// TIA Portal V17 export
// export: Created 2024-08-29T18:23:43.1204595Z, ExportSetting WithDefaults, DisplayName Totally Integrated Automation Portal, DisplayVersion V17 Update 7, DisplayName TIA Portal Openness, DisplayVersion V17 Update 7, DisplayName TIA Portal Version Control Interface, DisplayVersion V17, DisplayName SINAMICS Startdrive Advanced, DisplayVersion V17 SP2, DisplayName SINAMICS Startdrive G110M, G120, G120C, G120D, G120P, G115D, DisplayVersion V17 SP2, DisplayName SINAMICS Startdrive G130, G150, S120, S150, SINAMICS MV, S210, DisplayVersion V17 SP2, DisplayName STEP 7 Professional, DisplayVersion V17 Update 7, DisplayName STEP 7 Safety, DisplayVersion V17 Update 6, DisplayName WinCC Advanced / Unified PC, DisplayVersion V17 Update 7
DATA_BLOCK "inputs"   // DB1
{ S7_Optimized_Access := 'TRUE' }
VERSION : 0.1
// stored: AutoNumber false, DBAccessibleFromOPCUA true, DBAccessibleFromWebserver true, IsOnlyStoredInLoadMemory false, IsRetainMemResEnabled false, IsWriteProtectedInAS false, MemoryReserve 100
   VAR RETAIN
      inputSequence : Array[0..32, 0..25] of DInt;   // 32 entradas [modelo, paso]
   END_VAR
   VAR
      activeInputsReq : Array[0..31] of Bool;
   END_VAR
   VAR RETAIN
      maskSequence : Array[0..32, 0..25] of DInt;   // Máscara de entradas
   END_VAR
   VAR
      activeMask : Array[0..31] of Bool;
   END_VAR
   VAR RETAIN
      inputText : Array[0..31] of String;   // Texto HMI de cada entrada
   END_VAR
   VAR
      buttonStatus : Array[0..63] of Bool;
      activeInputsReqDInt : DInt := 131392;   // Estado de sensores en directo
      inputActive : Array[0..31] of Bool;
      euchnerReading : Array[0..254] of Char;
      nestScannerReading : String := '';
      upperScannerReading : String := '';
      nestScanerReceived : Array[0..254] of Char;
      nestScanerReceivedString : String := '';
      upperScannerReceived : Array[0..254] of Char;
      upperScannerReceivedString : String := '';
      euchnerReadingString : String := '$01';
      laserReading : Word := 16#0000;
      laserConstant : Real := 0.0005802801;
      laserReadingInt : DInt := 0;
      readingConversion : LReal := 0.0;
      euchnerName : String := '';
      euchner : Array[0..257] of Byte;
   END_VAR
BEGIN
   inputSequence[0,0] := 23724353;
   inputSequence[0,1] := 827_518_278;
   inputSequence[0,2..4] := 44756294;
   inputSequence[0,5] := 1_252_650_334;
   inputSequence[0,6..7] := 1_118_432_670;
   inputSequence[0,8] := 1_118_432_414;
   inputSequence[0,9] := 44690590;
   inputSequence[0,10] := 44892160;
   inputSequence[0,11..25] := 0;
   inputSequence[1,0] := 23724353;
   inputSequence[1,1] := 827_518_278;
   inputSequence[1,2..4] := 44756294;
   inputSequence[1,5] := 1_252_650_334;
   inputSequence[1,6..7] := 1_118_432_670;
   inputSequence[1,8] := 1_118_432_414;
   inputSequence[1,9] := 44690590;
   inputSequence[1,10] := 44892160;
   inputSequence[1,11..25] := 0;
   inputSequence[2,0] := 23724353;
   inputSequence[2,1] := 827_514_182;
   inputSequence[2,2..4] := 44752198;
   inputSequence[2,5] := 1_252_646_238;
   inputSequence[2,6..7] := 1_118_428_574;
   inputSequence[2,8] := 1_118_428_318;
   inputSequence[2,9] := 44686494;
   inputSequence[2,10] := 44892160;
   inputSequence[2,11..25] := 0;
   inputSequence[3,0] := 23724353;
   inputSequence[3,1] := 827_518_278;
   inputSequence[3,2..4] := 44756294;
   inputSequence[3,5] := 1_252_650_334;
   inputSequence[3,6..8] := 1_118_432_670;
   inputSequence[3,9] := 1_118_432_414;
   inputSequence[3,10] := 44690590;
   inputSequence[3,11] := 44892160;
   inputSequence[3,12..25] := 0;
   inputSequence[4,0] := 23724353;
   inputSequence[4,1] := 827_514_182;
   inputSequence[4,2..4] := 44752198;
   inputSequence[4,5] := 1_252_646_238;
   inputSequence[4,6..7] := 1_118_428_574;
   inputSequence[4,8] := 1_118_428_446;
   inputSequence[4,9] := 1_118_428_318;
   inputSequence[4,10] := 44686494;
   inputSequence[4,11] := 44892160;
   inputSequence[4,12..25] := 0;
   inputSequence[5,0..1] := 64;
   inputSequence[5,2..3] := 128;
   inputSequence[5,4..25] := 0;
   inputSequence[6,0] := 23724353;
   inputSequence[6,1] := 827_780_422;
   inputSequence[6,2] := 44756294;
   inputSequence[6,3] := 44755974;
   inputSequence[6,4] := 1_252_650_334;
   inputSequence[6,5..7] := 1_118_432_670;
   inputSequence[6,8] := 1_118_432_414;
   inputSequence[6,9] := 44630336;
   inputSequence[6,10..25] := 0;
   inputSequence[7,0] := 23724353;
   inputSequence[7,1] := 827_780_422;
   inputSequence[7,2] := 44756294;
   inputSequence[7,3] := 44755974;
   inputSequence[7,4] := 1_252_650_334;
   inputSequence[7,5..7] := 1_118_432_670;
   inputSequence[7,8] := 1_118_432_414;
   inputSequence[7,9] := 44630336;
   inputSequence[7,10..25] := 0;
   inputSequence[8,0] := 23724353;
   inputSequence[8,1] := 827_776_326;
   inputSequence[8,2] := 44752198;
   inputSequence[8,3] := 44751878;
   inputSequence[8,4] := 1_252_646_238;
   inputSequence[8,5] := 1_118_428_574;
   inputSequence[8,6] := 1_118_428_318;
   inputSequence[8,7] := 1_118_428_574;
   inputSequence[8,8] := 1_118_428_318;
   inputSequence[8,9] := 44630336;
   inputSequence[8,10..25] := 0;
   inputSequence[9,0] := 321;
   inputSequence[9,1] := 4193656;
   inputSequence[9,2] := 2_017_459_576;
   inputSequence[9,3] := 1_077_935_482;
   inputSequence[9,4] := 1_073_745_282;
   inputSequence[9,5..6] := 1_073_745_538;
   inputSequence[9,7..9] := 320;
   inputSequence[9,10..25] := 0;
   inputSequence[10,0] := 321;
   inputSequence[10,1] := 4193656;
   inputSequence[10,2] := 2_017_459_576;
   inputSequence[10,3] := 1_077_935_482;
   inputSequence[10,4] := 1_073_745_282;
   inputSequence[10,5..6] := 1_073_745_538;
   inputSequence[10,7..9] := 320;
   inputSequence[10,10..25] := 0;
   inputSequence[11,0] := 321;
   inputSequence[11,1] := 4193656;
   inputSequence[11,2] := 2_017_459_576;
   inputSequence[11,3] := 1_077_935_482;
   inputSequence[11,4] := 1_073_745_282;
   inputSequence[11,5..6] := 1_073_745_538;
   inputSequence[11,7..9] := 320;
   inputSequence[11,10..25] := 0;
   inputSequence[12,0] := 321;
   inputSequence[12,1] := 8387960;
   inputSequence[12,2] := 2_021_653_880;
   inputSequence[12,3] := 1_082_129_786;
   inputSequence[12,4] := 1_077_939_586;
   inputSequence[12,5] := 1_077_939_842;
   inputSequence[12,6] := 1_073_745_538;
   inputSequence[12,7..9] := 320;
   inputSequence[12,10..25] := 0;
   inputSequence[13,0] := 321;
   inputSequence[13,1] := 4193656;
   inputSequence[13,2] := 2_017_459_576;
   inputSequence[13,3] := 1_077_935_482;
   inputSequence[13,4] := 1_073_745_282;
   inputSequence[13,5..6] := 1_073_745_538;
   inputSequence[13,7..9] := 320;
   inputSequence[13,10..25] := 0;
   inputSequence[14,0] := 321;
   inputSequence[14,1] := 4193656;
   inputSequence[14,2] := 2_017_459_576;
   inputSequence[14,3] := 1_077_935_482;
   inputSequence[14,4] := 1_073_745_282;
   inputSequence[14,5..6] := 1_073_745_538;
   inputSequence[14,7..9] := 320;
   inputSequence[14,10..25] := 0;
   inputSequence[15,0] := 11;
   inputSequence[15,1] := 63040522;
   inputSequence[15,2] := 1_338_108_938;
   inputSequence[15,3] := 65137674;
   inputSequence[15,4] := 65135628;
   inputSequence[15,5] := 65134612;
   inputSequence[15,6] := 57344;
   inputSequence[15,7] := 805_363_712;
   inputSequence[15,8] := 10;
   inputSequence[15,9..25] := 0;
   inputSequence[16,0] := 321;
   inputSequence[16,1] := 8387960;
   inputSequence[16,2] := 2_021_653_880;
   inputSequence[16,3] := 1_082_129_786;
   inputSequence[16,4] := 1_077_939_586;
   inputSequence[16,5] := 1_077_939_842;
   inputSequence[16,6] := 1_073_745_538;
   inputSequence[16,7..9] := 320;
   inputSequence[16,10..25] := 0;
   inputSequence[17,0] := 321;
   inputSequence[17,1] := 4193656;
   inputSequence[17,2] := 2_017_459_576;
   inputSequence[17,3] := 1_077_935_482;
   inputSequence[17,4] := 1_073_745_282;
   inputSequence[17,5..6] := 1_073_745_538;
   inputSequence[17,7..9] := 320;
   inputSequence[17,10..25] := 0;
   inputSequence[18,0] := 321;
   inputSequence[18,1] := 4193656;
   inputSequence[18,2] := 2_017_459_576;
   inputSequence[18,3] := 1_077_935_482;
   inputSequence[18,4] := 1_073_745_282;
   inputSequence[18,5..6] := 1_073_745_538;
   inputSequence[18,7..9] := 320;
   inputSequence[18,10..25] := 0;
   inputSequence[19,0] := 321;
   inputSequence[19,1] := 4193656;
   inputSequence[19,2] := 2_017_459_576;
   inputSequence[19,3] := 1_077_935_482;
   inputSequence[19,4] := 1_073_745_282;
   inputSequence[19,5..6] := 1_073_745_538;
   inputSequence[19,7..9] := 320;
   inputSequence[19,10..25] := 0;
   inputSequence[20,0..25] := 0;
   inputSequence[21,0..25] := 0;
   inputSequence[22,0..25] := 0;
   inputSequence[23,0..25] := 0;
   inputSequence[24,0..25] := 0;
   inputSequence[25,0..25] := 0;
   inputSequence[26,0..25] := 0;
   inputSequence[27,0..25] := 0;
   inputSequence[28,0..25] := 0;
   inputSequence[29,0..25] := 0;
   inputSequence[30,0..25] := 0;
   inputSequence[31,0..25] := 0;
   inputSequence[32,0..25] := 0;
   activeInputsReq[0] := TRUE;
   activeInputsReq[1..5] := FALSE;
   activeInputsReq[6] := TRUE;
   activeInputsReq[7] := FALSE;
   activeInputsReq[8] := TRUE;
   activeInputsReq[9..16] := FALSE;
   activeInputsReq[17] := TRUE;
   activeInputsReq[18] := FALSE;
   activeInputsReq[19] := TRUE;
   activeInputsReq[20] := FALSE;
   activeInputsReq[21..22] := TRUE;
   activeInputsReq[23] := FALSE;
   activeInputsReq[24] := TRUE;
   activeInputsReq[25..31] := FALSE;
   maskSequence[0,0] := 66859008;
   maskSequence[0,1] := 66846720;
   maskSequence[0,2] := 66847168;
   maskSequence[0,3..4] := 66846848;
   maskSequence[0,5..8] := 66846720;
   maskSequence[0,9] := 66846862;
   maskSequence[0,10] := 66649232;
   maskSequence[0,11..25] := 0;
   maskSequence[1,0] := 66859008;
   maskSequence[1,1] := 66846720;
   maskSequence[1,2] := 66847168;
   maskSequence[1,3..4] := 66846848;
   maskSequence[1,5..8] := 66846720;
   maskSequence[1,9] := 66846862;
   maskSequence[1,10] := 66649232;
   maskSequence[1,11..25] := 0;
   maskSequence[2,0] := 66859008;
   maskSequence[2,1] := 66846720;
   maskSequence[2,2] := 66847168;
   maskSequence[2,3..4] := 66846848;
   maskSequence[2,5..8] := 66846720;
   maskSequence[2,9] := 66846862;
   maskSequence[2,10] := 66649232;
   maskSequence[2,11..25] := 0;
   maskSequence[3,0] := 66859008;
   maskSequence[3,1] := 66846720;
   maskSequence[3,2] := 66847168;
   maskSequence[3,3..4] := 66846848;
   maskSequence[3,5..7] := 66846720;
   maskSequence[3,8] := 66846976;
   maskSequence[3,9] := 66846720;
   maskSequence[3,10] := 66846848;
   maskSequence[3,11] := 66649232;
   maskSequence[3,12..25] := 0;
   maskSequence[4,0] := 66859008;
   maskSequence[4,1] := 66846720;
   maskSequence[4,2] := 66847168;
   maskSequence[4,3..4] := 66846848;
   maskSequence[4,5..7] := 66846720;
   maskSequence[4,8] := 66847168;
   maskSequence[4,9] := 66846720;
   maskSequence[4,10] := 66846848;
   maskSequence[4,11] := 66649232;
   maskSequence[4,12..25] := 0;
   maskSequence[5,0..1] := -65;
   maskSequence[5,2..3] := -129;
   maskSequence[5,4..25] := 0;
   maskSequence[6,0..2] := 66846720;
   maskSequence[6,3] := 66847168;
   maskSequence[6,4..8] := 66846720;
   maskSequence[6,9] := 66847168;
   maskSequence[6,10..25] := 0;
   maskSequence[7,0..1] := 66846720;
   maskSequence[7,2..3] := 66847168;
   maskSequence[7,4..6] := 66846720;
   maskSequence[7,7] := 66846976;
   maskSequence[7,8] := 66846720;
   maskSequence[7,9] := 66847168;
   maskSequence[7,10..25] := 0;
   maskSequence[8,0..1] := 66846720;
   maskSequence[8,2..3] := 66847168;
   maskSequence[8,4..5] := 66846720;
   maskSequence[8,6..7] := 66846976;
   maskSequence[8,8] := 66846720;
   maskSequence[8,9] := 66847168;
   maskSequence[8,10..25] := 0;
   maskSequence[9,0] := -322;
   maskSequence[9,1] := 2_014_248_960;
   maskSequence[9,2..3] := 983040;
   maskSequence[9,4..5] := 79687736;
   maskSequence[9,6] := 134_213_948;
   maskSequence[9,7..8] := -2;
   maskSequence[9,9] := 134_217_406;
   maskSequence[9,10..25] := 0;
   maskSequence[10,0] := -322;
   maskSequence[10,1] := 2_014_289_920;
   maskSequence[10,2..3] := 1024000;
   maskSequence[10,4..5] := 79687736;
   maskSequence[10,6] := 134_213_948;
   maskSequence[10,7..8] := -2;
   maskSequence[10,9] := 134_217_406;
   maskSequence[10,10..25] := 0;
   maskSequence[11,0] := -322;
   maskSequence[11,1] := 2_014_248_960;
   maskSequence[11,2..3] := 983040;
   maskSequence[11,4..5] := 79687736;
   maskSequence[11,6] := 134_213_948;
   maskSequence[11,7..8] := -2;
   maskSequence[11,9] := 134_217_406;
   maskSequence[11,10..25] := 0;
   maskSequence[12,0] := -322;
   maskSequence[12,1] := 2_014_248_960;
   maskSequence[12,2..3] := 983040;
   maskSequence[12,4..5] := 79687736;
   maskSequence[12,6] := 134_213_948;
   maskSequence[12,7..8] := -2;
   maskSequence[12,9] := 134_217_406;
   maskSequence[12,10..25] := 0;
   maskSequence[13,0] := -322;
   maskSequence[13,1] := 2_014_248_960;
   maskSequence[13,2..3] := 983040;
   maskSequence[13,4..5] := 79687736;
   maskSequence[13,6] := 134_213_948;
   maskSequence[13,7..8] := -2;
   maskSequence[13,9] := 134_217_406;
   maskSequence[13,10..25] := 0;
   maskSequence[14,0] := -322;
   maskSequence[14,1] := 2_014_248_960;
   maskSequence[14,2] := 806_289_408;
   maskSequence[14,3] := 983040;
   maskSequence[14,4..5] := 79687736;
   maskSequence[14,6] := 134_213_948;
   maskSequence[14,7..8] := -2;
   maskSequence[14,9] := 134_217_406;
   maskSequence[14,10..25] := 0;
   maskSequence[15,0] := 0;
   maskSequence[15,1] := 2_080_374_784;
   maskSequence[15,2..3] := 805_306_368;
   maskSequence[15,4..5] := 868_220_928;
   maskSequence[15,6..7] := 268_435_452;
   maskSequence[15,8..25] := 0;
   maskSequence[16,0] := -322;
   maskSequence[16,1] := 2_014_248_960;
   maskSequence[16,2..3] := 983040;
   maskSequence[16,4..5] := 79687736;
   maskSequence[16,6] := 134_213_948;
   maskSequence[16,7..8] := -2;
   maskSequence[16,9] := 134_217_406;
   maskSequence[16,10..25] := 0;
   maskSequence[17,0] := -322;
   maskSequence[17,1] := 2_014_248_960;
   maskSequence[17,2..3] := 983040;
   maskSequence[17,4..5] := 79687736;
   maskSequence[17,6] := 134_213_948;
   maskSequence[17,7..8] := -2;
   maskSequence[17,9] := 134_217_406;
   maskSequence[17,10..25] := 0;
   maskSequence[18,0] := -322;
   maskSequence[18,1] := 2_014_248_960;
   maskSequence[18,2..3] := 983040;
   maskSequence[18,4..5] := 79687736;
   maskSequence[18,6] := 134_213_948;
   maskSequence[18,7..8] := -2;
   maskSequence[18,9] := 134_217_406;
   maskSequence[18,10..25] := 0;
   maskSequence[19,0] := -322;
   maskSequence[19,1] := 2_014_248_960;
   maskSequence[19,2..3] := 983040;
   maskSequence[19,4..5] := 79687736;
   maskSequence[19,6] := 134_213_948;
   maskSequence[19,7..8] := -2;
   maskSequence[19,9] := 134_217_406;
   maskSequence[19,10..25] := 0;
   maskSequence[20,0..25] := 0;
   maskSequence[21,0..25] := 0;
   maskSequence[22,0..25] := 0;
   maskSequence[23,0..25] := 0;
   maskSequence[24,0..25] := 0;
   maskSequence[25,0..25] := 0;
   maskSequence[26,0..25] := 0;
   maskSequence[27,0..25] := 0;
   maskSequence[28,0..25] := 0;
   maskSequence[29,0..25] := 0;
   maskSequence[30,0..25] := 0;
   maskSequence[31,0..25] := 0;
   maskSequence[32,0..25] := 0;
   activeMask[0..11] := FALSE;
   activeMask[12..13] := TRUE;
   activeMask[14..17] := FALSE;
   activeMask[18..25] := TRUE;
   activeMask[26..31] := FALSE;
   inputText[0] := 'CLEAR DATA';
   inputText[1] := 'Clamp izq. cerrado PRX18151';
   inputText[2] := 'Clamp der. cerrado PRX18150';
   inputText[3] := 'Clamp plastic bridge cerrado PRX19130';
   inputText[4] := 'Plastic bridge presente PRX19090';
   inputText[5] := 'Reserva';
   inputText[6] := 'Herramental izq. pos. inicio PRX18130';
   inputText[7] := 'Herramental izq pos trabajo PRX19091';
   inputText[8] := 'Herramental der. pos. inicio PRX18131';
   inputText[9] := 'Reserva';
   inputText[10] := 'Track 1 izq. presente PRX18090';
   inputText[11] := 'Track 1 der. presente PRX18110';
   inputText[12] := 'Tornillo track izq. PRX19110';
   inputText[13] := 'Tornillo track der. PRX19111';
   inputText[14] := 'Track 2 izq. presente PRX18091';
   inputText[15] := 'Track 2 der. presente PRX18111';
   inputText[16] := 'Posicion nido colocar track PRX19150';
   inputText[17] := 'Posicion nido ensamble varilla PRX19151';
   inputText[18] := 'Quitar pieza';
   inputText[19..26] := 'Reserva';
   inputText[27] := 'Escaner motor OK';
   inputText[28] := 'Escaner Track izq OK';
   inputText[29] := 'Escaner Track der OK';
   inputText[30] := 'Motor conectado ';
   inputText[31] := 'RESERVA';
   buttonStatus[0] := FALSE;
   buttonStatus[1..4] := TRUE;
   buttonStatus[5..6] := FALSE;
   buttonStatus[7] := TRUE;
   buttonStatus[8..9] := FALSE;
   buttonStatus[10..11] := TRUE;
   buttonStatus[12] := FALSE;
   buttonStatus[13..16] := TRUE;
   buttonStatus[17..18] := FALSE;
   buttonStatus[19] := TRUE;
   buttonStatus[20] := FALSE;
   buttonStatus[21] := TRUE;
   buttonStatus[22] := FALSE;
   buttonStatus[23] := TRUE;
   buttonStatus[24] := FALSE;
   buttonStatus[25] := TRUE;
   buttonStatus[26..32] := FALSE;
   buttonStatus[33..35] := TRUE;
   buttonStatus[36..38] := FALSE;
   buttonStatus[39] := TRUE;
   buttonStatus[40..49] := FALSE;
   buttonStatus[50..57] := TRUE;
   buttonStatus[58..63] := FALSE;
   inputActive[0..5] := FALSE;
   inputActive[6] := TRUE;
   inputActive[7] := FALSE;
   inputActive[8] := TRUE;
   inputActive[9..16] := FALSE;
   inputActive[17..18] := TRUE;
   inputActive[19..31] := FALSE;
   euchnerReading[0] := '$01';
   euchnerReading[1..127] := '$00';
   euchnerReading[128..254] := ' ';
   nestScanerReceived[0..254] := ' ';
   upperScannerReceived[0..254] := ' ';
   euchner[0..1] := 16#00;
   euchner[2] := 16#44;
   euchner[3..7] := 16#00;
   euchner[8..147] := 16#20;
   euchner[148..257] := 16#00;
END_DATA_BLOCK
